// TIA Portal V18 export
TYPE "LGasp_typeAssiAAA"
// stored: IsFailsafeCompliant false
   STRUCT
      stazione : Int;   // stazione di appartenenza
      nome : WString[20];   // nome asse
      nometrad : WString[20];   // nome tradotto
      qatt : LReal;   // quota attuale letta da PC
      qset : LReal;   // quota target calcolata da PC
      corr : LReal;   // correttore letto e scritto da PC
      oldcorr : LReal;   // correttore precedente alla modifica letto da PC
      target : LReal;   // target = quota calcolata + correttore letta da PC
      sts : Struct   // stati
         DM_ok { ExternalWritable := 'False'} : Bool;   // dati macchina ok
         peh : Bool;   // asse in peh
         fault : Bool;   // asse in errore generico
         fcpos { ExternalWritable := 'False'} : Bool;   // asse in finecorsa software positivo
         fcneg { ExternalWritable := 'False'} : Bool;   // asse in finecorsa software negativo
         hwpos { ExternalWritable := 'False'} : Bool;   // asse in finecorsa hardware positivo
         hwneg { ExternalWritable := 'False'} : Bool;   // asse in finecorsa hardware negativo
         b07 : Bool;
         b8 : Bool;
         b9 : Bool;
         b10 : Bool;
         b11 : Bool;
         b12 : Bool;
         b13 : Bool;
         b14 : Bool;
         b15 : Bool;
      END_STRUCT;
      sts_PC : Word;   // stati appoggiati a PC che legge la word
   END_STRUCT;
END_TYPE
